PROGRAM Systemparameter
VAR
END_VAR

// Lesen
	// Objektzustände
	GVL.Robot_State 		:= Anlage.UR5.P_State;
	GVL.Greifer_State 		:= Anlage.Gripper.P_State;
	GVL.Sensor_State 		:= 1;

// Zuweisen
	// Eigenschaften	
	Anlage.HEX_E.P_LimitValue 		:= GVL.eKraftLimitValue;
	Anlage.HEX_E.P_ErreichtValue 	:= GVL.eKraftErreichtValue;

END_PROGRAM

(* stored: Version 1.1.0.1
   POU Systemparameter: Id {af4a7020-976b-475d-9afa-9c7a00ca4ce9}, SpecialFunc None *)
